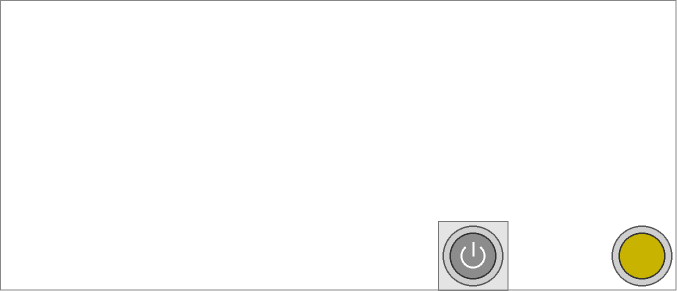
VISUALIZATION Visu  // 677x291
    PowerSwitch (438,221 70x70), variable: MAIN.bInput, behaviour: TOGGLE, style: Switch-PowerSwitch-Gray
    Lamp1 (607,221 70x70), variable: MAIN.bOutput, style: Lamp-Lamp1-Yellow
END_VISUALIZATION

(* stored: Version 1.1.0.1, ProductVersion 3.1.4024.12
   Visu Visu: Id {fd072645-4c5c-4b97-833e-8ad284fc89a9} *)
